// TIA Portal V17 export
// export: Created 2022-05-02T08:03:56.777081Z, ExportSetting WithDefaults, DisplayName Totally Integrated Automation Portal, DisplayVersion V17 Update 3, DisplayName TIA Portal Openness, DisplayVersion V17 Update 3, DisplayName TIA Portal Teamcenter Gateway, DisplayVersion V17 Update 3, DisplayName TIA Portal Version Control Interface, DisplayVersion V17, DisplayName SINAMICS Startdrive Advanced, DisplayVersion V17 Update2, DisplayName SINAMICS Startdrive G130, G150, S120, S150, SINAMICS MV, S210, DisplayVersion V17 Update2, DisplayName SINAMICS Startdrive G110M, G120, G120C, G120D, G120P, G115D, DisplayVersion V17 Update2, DisplayName STEP 7 Professional, DisplayVersion V17 Update 3, DisplayName STEP 7 CFC, DisplayVersion V17 Update 1, DisplayName STEP 7 Safety, DisplayVersion V17, DisplayName WinCC UA Professional, DisplayVersion V17 Update 3, DisplayName WinCC Unified Calendar, DisplayVersion V17, DisplayName WinCC Unified Performance Insight, DisplayVersion V17
FUNCTION "FC_CALCUL" : Void   // FC10, LAD
{ S7_Optimized_Access := 'TRUE' }
VERSION : 0.1
// stored: AutoNumber true, IsIECCheckEnabled false, SetENOAutomatically false, UDAEnableTagReadback false
   VAR_INPUT
      mon_entrée : Bool;
   END_VAR
   VAR CONSTANT
      PI : Real := 3.1416;
   END_VAR
BEGIN

REGION Network 1
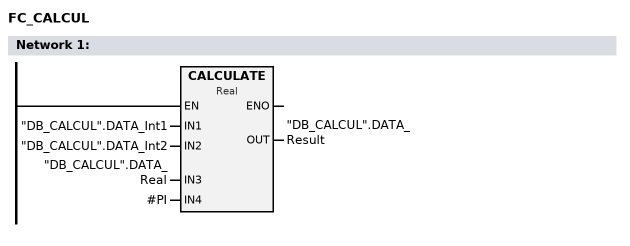
   RUNG wire#powerrail
      { S7_Templates := "SrcType := Real"; S7_Expression := "((IN1 / IN2)+IN3)*IN4" } Calculate(in1 := "DB_CALCUL".DATA_Int1, in2 := "DB_CALCUL".DATA_Int2, in3 := "DB_CALCUL".DATA_Real, in4 := #PI, out => "DB_CALCUL".DATA_Result)
   END_RUNG
   // the same network as SCL:
   "DB_CALCUL".DATA_Result := (("DB_CALCUL".DATA_Int1 / "DB_CALCUL".DATA_Int2)+"DB_CALCUL".DATA_Real)*#PI;
END_REGION

REGION Network 2 (SCL)
   IF "DB_CALCUL".DATA_Int1 <0  THEN
       "DB_CALCUL".DATA_Result := (("DB_CALCUL".DATA_Int1 / "DB_CALCUL".DATA_Int2) + "DB_CALCUL".DATA_Real) * #PI;
       ;
   END_IF;
END_REGION
END_FUNCTION
